PROGRAM Demo1
VAR_INPUT
	bExecute: BOOL;
	Rob: POINTER TO FB_1_ROB;
	SFCInit: BOOL;
END_VAR
VAR_OUTPUT
END_VAR
VAR
END_VAR

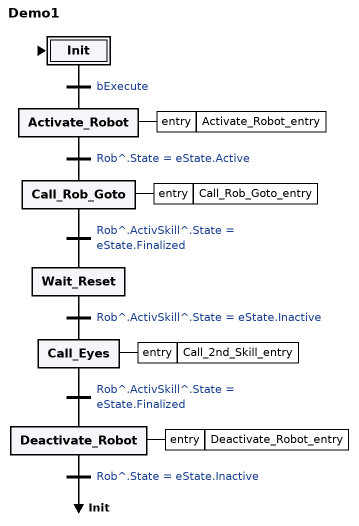
INITIAL_STEP Init:
END_STEP
TRANSITION FROM Init TO Activate_Robot
    := bExecute;
END_TRANSITION
STEP Activate_Robot:
    Activate_Robot_entry(P1);  // entry action
END_STEP
TRANSITION FROM Activate_Robot TO Call_Rob_Goto
    := Rob^.State = eState.Active;
END_TRANSITION
STEP Call_Rob_Goto:
    Call_Rob_Goto_entry(P1);  // entry action
END_STEP
TRANSITION FROM Call_Rob_Goto TO Wait_Reset
    := Rob^.ActivSkill^.State = eState.Finalized;
END_TRANSITION
STEP Wait_Reset:
END_STEP
TRANSITION FROM Wait_Reset TO Call_Eyes
    := Rob^.ActivSkill^.State = eState.Inactive;
END_TRANSITION
STEP Call_Eyes:
    Call_2nd_Skill_entry(P1);  // entry action
END_STEP
TRANSITION FROM Call_Eyes TO Deactivate_Robot
    := Rob^.ActivSkill^.State = eState.Finalized;
END_TRANSITION
STEP Deactivate_Robot:
    Deactivate_Robot_entry(P1);  // entry action
END_STEP
TRANSITION FROM Deactivate_Robot TO Init
    := Rob^.State = eState.Inactive;
END_TRANSITION

ACTION Activate_Robot_entry:
Rob^.Activate();
END_ACTION

ACTION Call_2nd_Skill_entry:
ROB^.Skills[2]^.Execute();
END_ACTION

ACTION Call_Rob_Goto_entry:
Rob^.Skills[1]^.Execute();
END_ACTION

ACTION Deactivate_Robot_entry:
Rob^.Deactivate();
END_ACTION

END_PROGRAM

(* stored: Version 1.1.0.1, ProductVersion 3.1.4026.18
   POU Demo1: Id {91af6b76-831c-43b6-9c52-2ccba4bf085a}, SpecialFunc None
   Action Activate_Robot_entry: Id {cb2f0cf5-7f9a-4846-91f6-fb59c90389d8}
   Action Call_2nd_Skill_entry: Id {71902e93-ed0b-4c27-91d3-25303768aa84}
   Action Call_Rob_Goto_entry: Id {d0acbf1c-0b96-427e-82dd-7405bcf4bc3e}
   Action Deactivate_Robot_entry: Id {4998cc69-d166-44b6-9940-8fb589f630e3} *)
